// Mitsubishi GX Works2 project: extracted manufa example   PLC: FX3U/FX3UC

PROGRAM MAIN
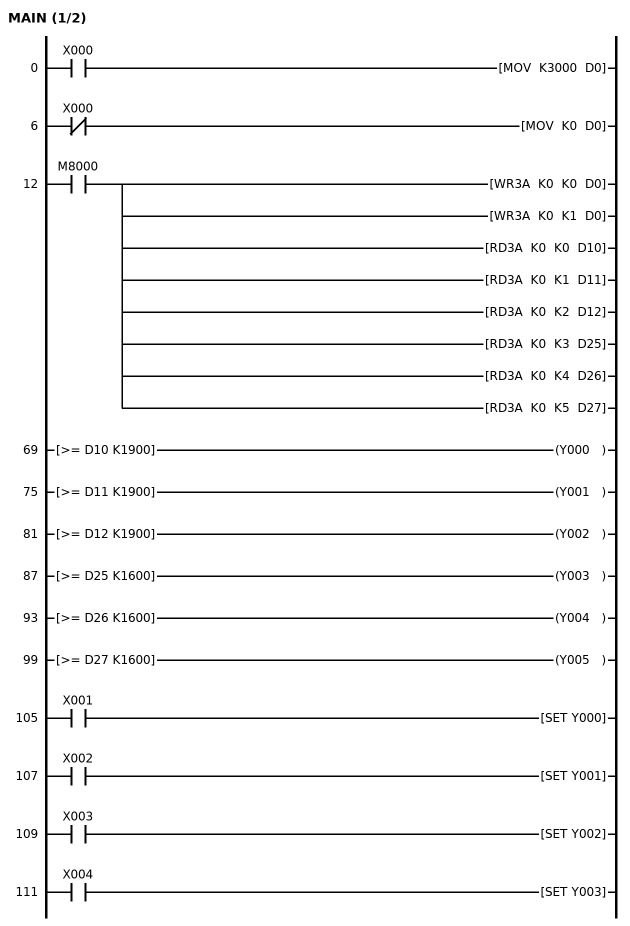
0     LD      X000
      MOV     K3000 D0
6     LDI     X000
      MOV     K0 D0
12    LD      M8000
      WR3A    K0 K0 D0
      WR3A    K0 K1 D0
      RD3A    K0 K0 D10
      RD3A    K0 K1 D11
      RD3A    K0 K2 D12
      RD3A    K0 K3 D25
      RD3A    K0 K4 D26
      RD3A    K0 K5 D27
69    LD>=    D10 K1900
      OUT     Y000
75    LD>=    D11 K1900
      OUT     Y001
81    LD>=    D12 K1900
      OUT     Y002
87    LD>=    D25 K1600
      OUT     Y003
93    LD>=    D26 K1600
      OUT     Y004
99    LD>=    D27 K1600
      OUT     Y005
105   LD      X001
      SET     Y000
107   LD      X002
      SET     Y001
109   LD      X003
      SET     Y002
111   LD      X004
      SET     Y003
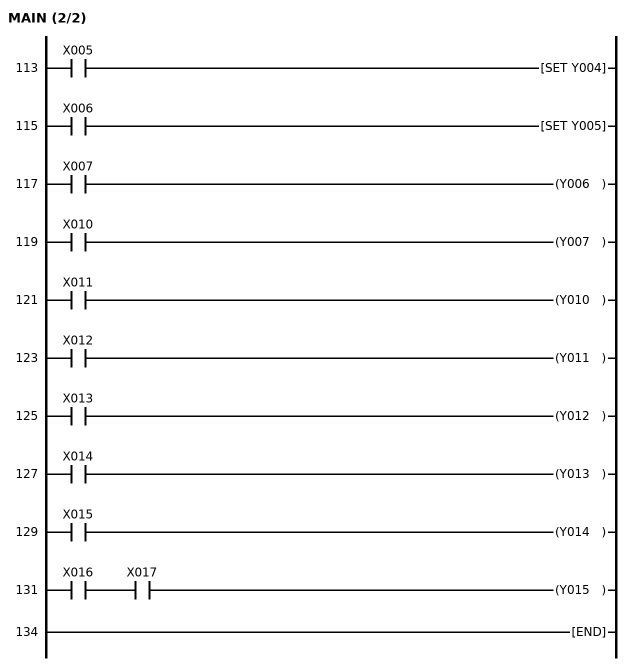
113   LD      X005
      SET     Y004
115   LD      X006
      SET     Y005
117   LD      X007
      OUT     Y006
119   LD      X010
      OUT     Y007
121   LD      X011
      OUT     Y010
123   LD      X012
      OUT     Y011
125   LD      X013
      OUT     Y012
127   LD      X014
      OUT     Y013
129   LD      X015
      OUT     Y014
131   LD      X016
      AND     X017
      OUT     Y015
134   END
END_PROGRAM
